{attribute 'linkalways'} 
{attribute 'no_explicit_call' := 'This FB is a CLASS and must be accessed using methods or properties'}
{attribute 'enable_dynamic_creation'}
FUNCTION_BLOCK FINAL Node_LREAL_TO_DINT EXTENDS Node
VAR
	in : _LREAL(0.0);
	out : _DINT(0);
	success : _BOOL(FALSE);
END_VAR

METHOD PUBLIC  Clone : I_Node
VAR
	pNode : POINTER TO Node_LREAL_TO_DINT;
END_VAR
pNode := __NEW(Node_LREAL_TO_DINT);
Clone := pNode^;
END_METHOD

METHOD FB_init : BOOL
VAR_INPUT
	bInitRetains : BOOL; // if TRUE, the retain variables are initialized (warm start / cold start)
	bInCopyCode : BOOL;  // if TRUE, the instance afterwards gets moved into the copy code (online change)
END_VAR
AddParameter('in', in);
AddOutput('out', out);
AddOutput('success', success);

this^.Metadatum.AddBoolAsMetadata('deprecated', true);
END_METHOD

METHOD PROTECTED OnExecute
VAR
END_VAR
success.Value := TryConvert_LREAL_TO_DINT(in.Value, out.Value);
END_METHOD

END_FUNCTION_BLOCK

(* stored: Version 1.1.0.1, ProductVersion 3.1.4026.18
   POU Node_LREAL_TO_DINT: Id {5bd06af0-f4f3-030e-2b9e-27e68e2098ad}, SpecialFunc None
   Folder Constructor: Id {12e0d75b-48d3-0a5e-13eb-ee5de9186166}
   Method Clone: Id {98715d79-b82d-0b50-109a-9b0629282442}
   Method FB_init: Id {1e3ca0c4-8b73-0fcf-2018-7a64900198c4}
   Method OnExecute: Id {6bbe4b2f-29bd-032d-180b-62570a1e7954} *)
